Yaskawa INFORM job: ABOVE-TO-BELOW.JBI

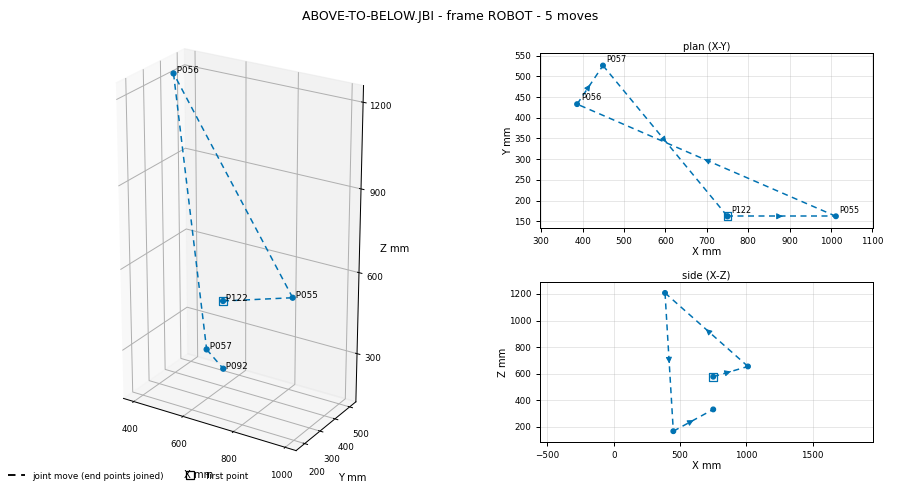
[picture p0: tool path of ABOVE-TO-BELOW.JBI in frame ROBOT, 5 of 5 moves have a stored position in this frame; points joined in program order, loops and branches not executed]
/JOB
//NAME ABOVE-TO-BELOW
///FOLDERNAME FOLDER001
//POS
///NPOS 0,0,0,5,0,0
///TOOL 1
///POSTYPE ROBOT
///RECTAN
///RCONF 0,0,0,0,0,0,0,0,0,0,0,0,0,0,0,0,0,0,0,0,0,0,0,0
P00055=1011.893,162.000,653.762,180.0000,-45.0000,0.0000
P00056=386.675,432.866,1207.867,11.5117,-39.6988,90.4579
P00057=449.192,526.165,165.762,5.4296,56.9271,40.1006
P00092=750.003,161.812,330.004,0.1640,10.0066,0.1393
///RCONF 1,0,0,0,0,0,0,0,0,0,0,0,0,0,0,0,0,0,0,0,0,0,0,0
P00122=750.004,162.000,576.437,180.0000,-9.9968,0.0000
//INST
///DATE 2025/09/30 16:24
///ATTR SC,RW
///GROUP1 RB1
NOP
MOVJ P122 VJ=100.00 PL=3
MOVJ P055 VJ=100.00 PL=3
MOVJ P056 VJ=100.00 PL=3
MOVJ P057 VJ=100.00 PL=3
MOVJ P092 VJ=100.00 PL=3
END
